FUNCTION_BLOCK AutoResetCdt (* CAT Function Block Type *)
  (* Standard: 61499-2 *)
  (* Version 0.0, 8/3/2026, Schneider Electric, template *)
  PACKAGE SE.Nereda;
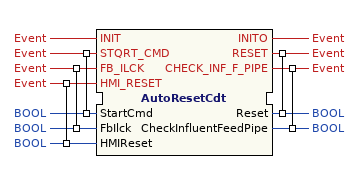
  EVENT_INPUT
    INIT; (* Initialization Request *)
    STQRT_CMD WITH StartCmd;
    FB_ILCK WITH FbIlck;
    HMI_RESET WITH HMIReset;
  END_EVENT
  EVENT_OUTPUT
    INITO; (* Initialization Confirm *)
    RESET WITH Reset;
    CHECK_INF_F_PIPE WITH CheckInfluentFeedPipe;
  END_EVENT
  VAR_INPUT
    StartCmd : BOOL;
    FbIlck : BOOL;
    HMIReset : BOOL;
  END_VAR
  VAR_OUTPUT
    Reset : BOOL;
    CheckInfluentFeedPipe : BOOL;
  END_VAR
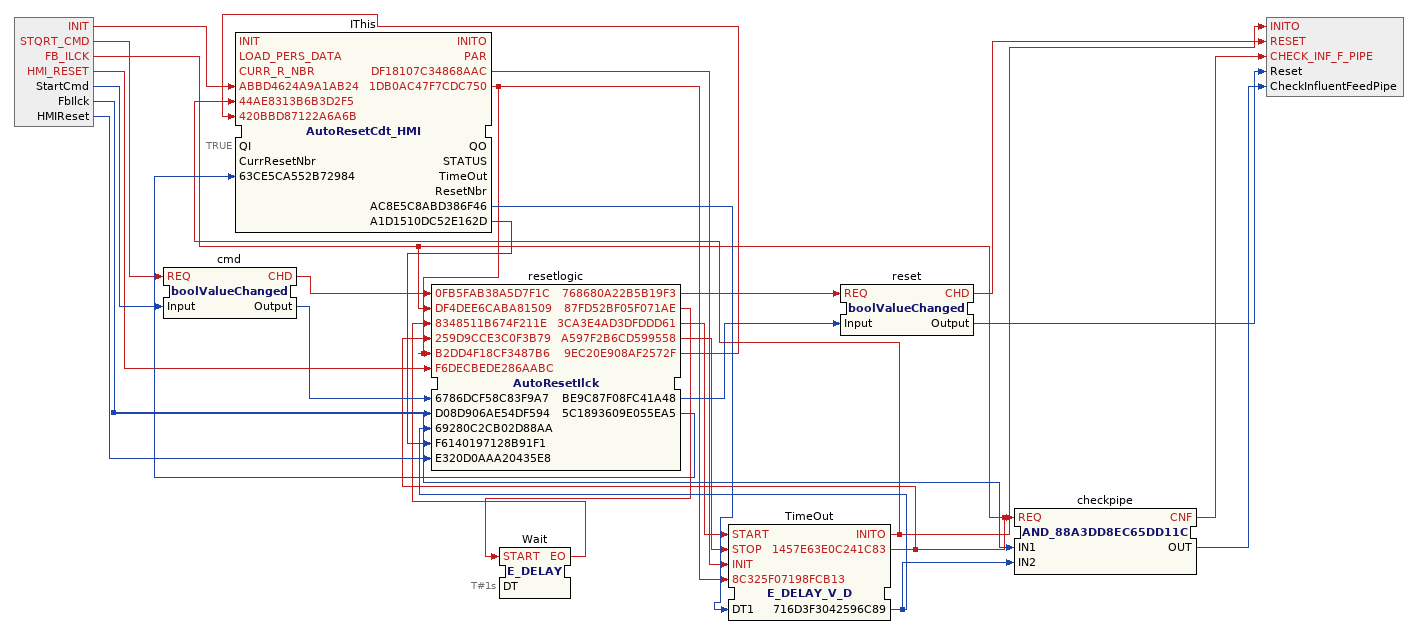
  FBS
    IThis : AutoResetCdt_HMI(QI := TRUE);
    resetlogic : AutoResetIlck;
    reset : boolValueChanged;
    cmd : boolValueChanged;
    Wait : E_DELAY(DT := T#1s);
    TimeOut : E_DELAY_V_D;
    checkpipe : AND_88A3DD8EC65DD11C; {SET_ATTRIBUTE(Configuration.GenericFBType.InterfaceParams, Runtime.Standard#CNT:=2;OUT:BOOL)}
  END_FBS
  EVENT_CONNECTIONS
    resetlogic.768680A22B5B19F3 TO reset.REQ;
    reset.CHD TO RESET;
    cmd.CHD TO resetlogic.0FB5FAB38A5D7F1C;
    STQRT_CMD TO cmd.REQ;
    FB_ILCK TO resetlogic.DF4DEE6CABA81509;
    resetlogic.87FD52BF05F071AE TO Wait.START;
    Wait.EO TO resetlogic.8348511B674F211E;
    TimeOut.INITO TO INITO;
    TimeOut.1457E63E0C241C83 TO resetlogic.259D9CCE3C0F3B79;
    resetlogic.3CA3E4AD3DFDDD61 TO TimeOut.START;
    resetlogic.A597F2B6CD599558 TO TimeOut.STOP;
    checkpipe.CNF TO CHECK_INF_F_PIPE;
    FB_ILCK TO checkpipe.REQ;
    TimeOut.1457E63E0C241C83 TO checkpipe.REQ;
    INIT TO IThis.ABBD4624A9A1AB24;
    TimeOut.INITO TO IThis.44AE8313B6B3D2F5;
    resetlogic.9EC20E908AF2572F TO IThis.420BBD87122A6A6B;
    IThis.DF18107C34868AAC TO TimeOut.INIT;
    IThis.1DB0AC47F7CDC750 TO resetlogic.B2DD4F18CF3487B6;
    IThis.1DB0AC47F7CDC750 TO TimeOut.8C325F07198FCB13;
    HMI_RESET TO resetlogic.F6DECBEDE286AABC;
  END_CONNECTIONS
  DATA_CONNECTIONS
    resetlogic.BE9C87F08FC41A48 TO reset.Input;
    reset.Output TO Reset;
    cmd.Output TO resetlogic.6786DCF58C83F9A7;
    StartCmd TO cmd.Input;
    FbIlck TO resetlogic.D08D906AE54DF594;
    TimeOut.716D3F3042596C89 TO resetlogic.69280C2CB02D88AA;
    checkpipe.OUT TO CheckInfluentFeedPipe;
    FbIlck TO checkpipe.IN1;
    TimeOut.716D3F3042596C89 TO checkpipe.IN2;
    IThis.AC8E5C8ABD386F46 TO TimeOut.DT1;
    IThis.A1D1510DC52E162D TO resetlogic.F6140197128B91F1;
    resetlogic.5C1893609E055EA5 TO IThis.63CE5CA552B72984;
    HMIReset TO resetlogic.E320D0AAA20435E8;
  END_CONNECTIONS
END_FUNCTION_BLOCK
